DATA_BLOCK "Global-DB"
{ S7_Optimized_Access := 'TRUE' }
VERSION : 0.1
NON_RETAIN
   VAR
      Vorlauftemperatur : Real;
      Ruecklauftemperatur : Real;
      Auto : Bool;
   END_VAR


BEGIN
   Auto := true;

END_DATA_BLOCK

